FUNCTION_BLOCK fBPulse1s
VAR_OUTPUT
	xFlanco: BOOL;
	xOut: BOOL;
END_VAR
VAR
	tTempo: Ton;
	iSeg: UDINT;
	pPulse: R_trig;
	iSeg_Ant: UDINT;
	PULSO: BLINK;
END_VAR



tTempo(IN:=NOT(tTempo.Q) , PT:=T#7D );
iSeg:=TIME_TO_DWORD(tTempo.ET)/1000;
pPulse(CLK:= (iSeg>iSeg_Ant) );
iSeg_Ant:=iSeg;

xFlanco:=pPulse.Q;

PULSO(ENABLE:= TRUE, TIMELOW:= T#1S, TIMEHIGH:= T#1S, OUT=> xOut);

END_FUNCTION_BLOCK

(* stored: Version 1.1.0.1, ProductVersion 3.1.4024.10
   POU fBPulse1s: Id {335d8a60-21d8-409e-bbf0-7fbe0a60ed72}, SpecialFunc None *)
